(* IEC 61131-3 sources: moqui-plc/simatic-ax/src/moqui/framework/src/main/org/moqui/util, 6 files *)

(* ---- Clocks.st ---- *)
(* Generated clocks for timing generation *)
TYPE Clocks : STRUCT
	(*
     * SystemClock is the main high-speed clock, e.g., from the task cycle.
     * All other clocks are derived from it.
     *)
    systemClock : BOOL; (* Main system clock 100 Hz, duty-cycle 50% *)
    (* Derived clock pulses (one-cycle TRUE). Derived from systemClock rising edge *)
    clock10ms : BOOL; (* 10ms pulse *)
    clock100ms : BOOL; (* 100ms pulse *)
    clock1s : BOOL; (* 1 second pulse *)
    clock1minute : BOOL; (* 1 minute pulse *)
	(* Extend based on your needs *)
END_STRUCT; END_TYPE

(* ---- MeanFilterType.st ---- *)
TYPE MeanFilterType : (
    SMA, (* Simple Moving Average *)
    WMA_Ramp, (* Weighted Moving Average, linear weights 1..N from oldest..newest (O(1)) *)
    WMA_Triangular, (* Symmetric triangular weights, center-weighted (O(N)) *)
    WMA_TriangularOddOnly, (* Symmetric triangular weights, requires odd windowSize (O(N)) *)
    TRI_SMA2, (* Triangular approximation via two SMA in cascade (O(1) per tick, extra memory) *)
    EMA (* Exponential Moving Average (alpha mandatory) *)
); END_TYPE

(* ---- nowTimestamp.st ---- *)
USING Siemens.Simatic.S71500.Clocks;

FUNCTION nowTimestamp : DATE_AND_TIME
	VAR
		localDateTime : LDATE_AND_TIME;
		execResult : WORD;
	END_VAR

	nowTimestamp := DT#1970-01-01-00:00:00;
	execResult := GetLocalDateTime(value => localDateTime);
	IF (execResult = WORD#16#0000) OR (execResult = WORD#16#0001) THEN
		nowTimestamp := TO_DT(localDateTime);
	END_IF;
	END_FUNCTION

(* ---- ClockGeneration.st ---- *)
FUNCTION_BLOCK ClockGeneration
VAR_EXTERNAL
    clks : Clocks;
END_VAR
VAR_INPUT
    operationType : OperatingMode;
END_VAR
VAR
    tick100ms : UDINT := UDINT#10;
    tick1s : UDINT := UDINT#10;
    tick1minute : UDINT := UDINT#60;
END_VAR

IF operationType = OperatingMode#Init THEN
    tick100ms := UDINT#10;
    tick1s := UDINT#10;
    tick1minute := UDINT#60;
END_IF;

clks.clock10ms := TRUE;

IF tick100ms > UDINT#1 THEN
    tick100ms := tick100ms - UDINT#1;
    clks.clock100ms := FALSE;
ELSE
    tick100ms := UDINT#10;
    clks.clock100ms := TRUE;
END_IF;

IF clks.clock100ms THEN
    IF tick1s > UDINT#1 THEN
        tick1s := tick1s - UDINT#1;
        clks.clock1s := FALSE;
    ELSE
        tick1s := UDINT#10;
        clks.clock1s := TRUE;
    END_IF;
ELSE
    clks.clock1s := FALSE;
END_IF;

IF clks.clock1s THEN
    IF tick1minute > UDINT#1 THEN
        tick1minute := tick1minute - UDINT#1;
        clks.clock1minute := FALSE;
    ELSE
        tick1minute := UDINT#60;
        clks.clock1minute := TRUE;
    END_IF;
ELSE
    clks.clock1minute := FALSE;
END_IF;
END_FUNCTION_BLOCK

(* ---- IIRFilter.st ---- *)
FUNCTION_BLOCK IIRFilter
	VAR_INPUT
	    execute : BOOL;
	    clock : BOOL;
	    reset : BOOL;
	    input : REAL;
	    T : REAL;
	    tickTime : TIME := T#10ms;
	END_VAR
	VAR_OUTPUT
	    output : REAL;
	    done : BOOL;
	    busy : BOOL;
	    error : BOOL;
	    errorId : INT;
	    timeElapsed : REAL;
	END_VAR
	VAR
	    init : BOOL;
	    elapsedTicks : UDINT;
	    deltaTime : REAL;
	    alpha : REAL;
	END_VAR

	(* Defaults *)
	done := FALSE;
	busy := FALSE;
	error := FALSE;
	errorId := 0;

	(* AX note: keep nominal 10 ms sampling for the first porting pass.
	 * This preserves the filter behavior much better than the old passthrough stub,
	 * while avoiding TIME conversions that this AX target does not currently accept. *)
	IF tickTime <= T#0S THEN
	    error := execute;
	    errorId := 1;
	    busy := FALSE;
	    RETURN;
	END_IF;

	deltaTime := REAL#0.01;

	IF reset THEN
	    init := FALSE;
	    elapsedTicks := UDINT#0;
	END_IF;

	IF execute THEN
	    busy := TRUE;

	    IF NOT init THEN
	        output := input;
	        init := TRUE;
	        elapsedTicks := UDINT#0;
	    ELSE
	        IF clock THEN
	            IF T > REAL#0.0 THEN
					IF T > deltaTime THEN
						alpha := deltaTime / T;
					ELSE
						alpha := REAL#1.0;
					END_IF;
	                output := output + alpha * (input - output);
	            ELSE
	                output := input;
	            END_IF;

	            elapsedTicks := elapsedTicks + UDINT#1;
	        END_IF;
	    END_IF;

	    timeElapsed := TO_REAL(elapsedTicks) * deltaTime;
	    done := NOT error;
	ELSE
	    busy := FALSE;
	    done := FALSE;
	    timeElapsed := REAL#0.0;
	END_IF;
END_FUNCTION_BLOCK

(* ---- SShapedFunc.st ---- *)
FUNCTION_BLOCK SShapedFunc
	VAR_INPUT
	    execute : BOOL;
	    clock : BOOL;
	    startValue : REAL;
	    endValue : REAL;
	    duration : TIME;
	    tickTime : TIME := T#10ms;
	END_VAR
	VAR_OUTPUT
	    output : REAL;
	    done : BOOL;
	    busy : BOOL;
	    error : BOOL;
	    errorId : INT;
	END_VAR
	VAR
	    prevExecute : BOOL;
	    active : BOOL;
	    elapsedTicks : UDINT;
	    totalTicks : UDINT;
	    progress : REAL;
	    deltaValue : REAL;
		remainingTime : TIME;
	END_VAR

	done := FALSE;
	busy := FALSE;
	error := (errorId <> 0);

	IF execute AND NOT prevExecute THEN
	    errorId := 0;
	    IF (duration <= T#0S) OR (tickTime <= T#0S) THEN
	        error := TRUE;
	        errorId := 1;
	        active := FALSE;
	    ELSE
	        active := TRUE;
	        elapsedTicks := UDINT#0;
			remainingTime := duration;
			totalTicks := UDINT#0;
			WHILE remainingTime > T#0S DO
				totalTicks := totalTicks + UDINT#1;
				IF remainingTime > tickTime THEN
					remainingTime := remainingTime - tickTime;
				ELSE
					remainingTime := T#0S;
				END_IF;
			END_WHILE;
	        IF totalTicks = UDINT#0 THEN
				totalTicks := UDINT#1;
			END_IF;

	        deltaValue := endValue - startValue;
	        output := startValue;
	    END_IF;
	END_IF;

	IF execute THEN
	    IF active THEN
	        busy := TRUE;

	        IF clock THEN
	            IF elapsedTicks < totalTicks THEN
	                elapsedTicks := elapsedTicks + UDINT#1;
	            END_IF;
	        END_IF;

	        progress := TO_REAL(elapsedTicks) / TO_REAL(totalTicks);

	        IF progress >= REAL#1.0 THEN
	            output := endValue;
	            active := FALSE;
	            done := TRUE;
	        ELSE
	            output := startValue + deltaValue * (REAL#3.0 * progress * progress - REAL#2.0 * progress * progress * progress);
	        END_IF;
	    ELSE
	        IF NOT error THEN
	            done := TRUE;
	        END_IF;
	    END_IF;
	ELSE
	    active := FALSE;
	    elapsedTicks := UDINT#0;
	    totalTicks := UDINT#0;
	    errorId := 0;
	END_IF;

	prevExecute := execute;
END_FUNCTION_BLOCK
